{attribute 'linkalways'} 
{attribute 'no_explicit_call' := 'This FB is a CLASS and must be accessed using methods or properties'}
{attribute 'enable_dynamic_creation'}
FUNCTION_BLOCK Node_F_VN_FillContainer_TcVnVector2_UINT EXTENDS VisionNode
VAR
    ipContainer : _ITcVnContainer;
    aValue : _TcVnVector2_UINT;
    hrPrev : _HRESULT(S_OK);
    hresult : _HRESULT(S_OK);
END_VAR

METHOD PUBLIC  Clone : I_Node
VAR
    pNode : POINTER TO Node_F_VN_FillContainer_TcVnVector2_UINT;
END_VAR
pNode := __NEW(Node_F_VN_FillContainer_TcVnVector2_UINT);
Clone := pNode^;
END_METHOD

METHOD FB_init : BOOL
VAR_INPUT
    bInitRetains : BOOL; // if TRUE, the retain variables are initialized (warm start / cold start)
    bInCopyCode : BOOL;  // if TRUE, the instance afterwards gets moved into the copy code (online change)
END_VAR
AddInput('ipContainer', ipContainer);
AddInput('aValue', aValue);
AddInput('hrPrev', hrPrev);
AddOutput('ipContainer', ipContainer);
AddOutput('hresult',hresult);
END_METHOD

METHOD PROTECTED OnExecute
hresult.Value := F_VN_FillContainer_TcVnVector2_UINT(
    ipContainer := ipContainer.Value,
    aValue := aValue.Value,
    hrPrev:= hrPrev.Value);
END_METHOD

METHOD PUBLIC PreExecutionCheck
VAR_INPUT
    Check : I_PreExecutionChecks;
END_VAR
Check.IsTrue(ipContainer.IsValid, 'ipContainer must be a valid container');
Check.IsTrue(ipContainer.IsType(TC_GLOBAL_CONST_LIST.ContainerType_Vector_TcVnVector2_UINT), 'ipContainer contains incorrect type');
END_METHOD

END_FUNCTION_BLOCK

(* stored: Version 1.1.0.1, ProductVersion 3.1.4026.13
   POU Node_F_VN_FillContainer_TcVnVector2_UINT: Id {d9183b5a-a577-4d25-ad3b-9a66cd36bdb1}, SpecialFunc None
   Folder Constructor: Id {9266e7c3-8fc9-4b4c-ad51-da316d2a91be}
   Method Clone: Id {06bd3509-6b68-4aaf-ba69-de2c2d30ae66}
   Method FB_init: Id {9395b744-dec3-40bd-b317-c12551757257}
   Method OnExecute: Id {9e815f76-723f-47d2-a5f2-606a5bfb1a41}
   Method PreExecutionCheck: Id {d64f223c-ad6a-4559-b471-d92806dfe75f} *)
